# EPICS substitutions: ek9000App/Db/EL4038.substitutions
file EL4038.template
{       pattern
        {
                TERMINAL,

        }
        {
        }
}
